// TIA Portal V19 export
FUNCTION "BTrk_Presence" : Void   // FC124, LAD
// stored: Access Published, SetENOAutomatically false
   VAR_INPUT
      Item : "BTrk_item";
   END_VAR
BEGIN

REGION Network 1 (SCL)
   ENO := #Item.B_ID <> 0;
END_REGION
END_FUNCTION
